FUNCTION_BLOCK FB_Observable_ULINT EXTENDS FB_AbstractObservable
VAR
    _nVal:              ULINT;
    _nOldVal:           ULINT;
END_VAR

METHOD FB_init : BOOL
VAR_INPUT
    bInitRetains:       BOOL; // if TRUE, the retain variables are initialized (warm start / cold start)
    bInCopyCode:        BOOL;  // if TRUE, the instance afterwards gets moved into the copy code (online change)
END_VAR
THIS^._nTypeClass := __SYSTEM.TYPE_CLASS.TYPE_ULINT;
END_METHOD

PROPERTY nDataSize : UDINT
GET
nDataSize := SIZEOF(LINT);
END_GET
END_PROPERTY

PROPERTY nValue64 : ULINT
GET
nValue64 := THIS^._nVal;
END_GET
SET
THIS^._nOldVal := THIS^._nVal;
THIS^._nVal := nValue64;

THIS^.NotifyWithConditions();
END_SET
END_PROPERTY

PROPERTY PROTECTED pData : POINTER TO BYTE
GET
pData := ADR(THIS^._nVal);
END_GET
END_PROPERTY

METHOD  ValueChanged : BOOL
VAR_INPUT
END_VAR
ValueChanged := THIS^._nOldVal <> THIS^._nVal;
END_METHOD

END_FUNCTION_BLOCK

(* stored: Version 1.1.0.1, ProductVersion 3.1.4024.12
   POU FB_Observable_ULINT: Id {7f91ecee-6834-01c7-1530-0b2a8fa1a37b}, SpecialFunc None
   Method FB_init: Id {97efe427-5c24-0e67-0dab-113dcb67bc16}
   Property nDataSize: Id {0366fbfb-317e-0543-2fec-72f372a9bdca}
   Get Get: Id {055934c7-6155-089e-281c-342017f4ca99}
   Property nValue64: Id {f8e95353-ec07-0230-32a2-a85a338193fb}
   Get Get: Id {0de93e6d-7a22-0f39-2de1-712b947c95d9}
   Set Set: Id {e74de1d8-dc64-0705-03cc-87532ce7f34b}
   Property pData: Id {1fe7a723-d2b7-081a-0fdc-74782f100faf}
   Get Get: Id {5d3ee7eb-2a5f-0885-2d09-d3735d523a72}
   Method ValueChanged: Id {85fa7587-27db-0a90-1b93-fc2aa3be7e55} *)
